# EPICS substitutions: mpgSupport/Db/ioc/evgPatternXL00.substitutions
file mpgEventAll.db
{
#                                  Check    Trigger
#          Device                PNET Data  Seq Ram
  pattern { DEVICE        , SYSI , CHECKI , SENDI  , SPEED                   }
          { IOC:IN20:EV01 , SYS0 ,   1    ,   1    , EVG:IN20:EV01:CTRL.R1SP }
}
file bsaEdefAll.db {
  pattern { DEVICE        , SYSI }
 	  { IOC:IN20:EV01 , SYS0 }
}
file evrPatternAll.db {
#	    Device        ,     Send Seq Ram
  pattern { DEVICE        ,         LINK4            , LINK5 , LINK6 , TREF }
	  { IOC:IN20:EV01 , IOC:IN20:EV01:SEQRAMSEND ,   ""  ,   ""  , 1E06 }
}
